// TIA Portal V20 export
DATA_BLOCK "ET200SP_201"   // DB227
// stored: MemoryReserve 100
   VAR
      "SP201.00 AUTO INITIATE PBL (GREEN)" : Bool;
      "SP201.01 STOP PBL (RED)" : Bool;
      SPARE1 : Bool;
      SPARE2 : Bool;
      SPARE3 : Bool;
      SPARE4 : Bool;
      SPARE5 : Bool;
      SPARE6 : Bool;
      "SP201.08 MAIN HMI POWER TRIPPED E110CB" : Bool;
      SPARE7 : Bool;
      SPARE8 : Bool;
      SPARE9 : Bool;
      SPARE10 : Bool;
      SPARE11 : Bool;
      SPARE12 : Bool;
      SPARE13 : Bool;
   END_VAR
BEGIN
END_DATA_BLOCK
